# EPICS substitutions: iocs/MC02/db/SAI_IOCsystem.substitutions
# DEVICE: device name
# CARD:
# CS_VERSION_VAL

file /opt/epics/modules/uIOCSystem/db/uIOCsystem.template {
pattern { DEVICE, CARD, CS_VERSION_VAL}
	{ "XF:06BM-OP{MC:02}", "0", "v0.01" }
}

#EOF
